// Mitsubishi GX Works2 project: Group13 - Copy   PLC: FX3G

// global labels: Global1
VAR_GLOBAL
  Start_of_Day AT X007 : BOOL;
  Y_0 AT Y000 : BOOL;
  Out_Of_Stock AT M1 : BOOL;
  Emergency_Button AT X005 : BOOL;
  Out_Of_Stock_Hold AT M2 : BOOL;
  Oats_Input AT D1100 : REAL;
  Honey_Input AT D1110 : REAL;
  Protein_Input AT D1120 : REAL;
  Oats_Quantity AT D1130 : REAL;
  Honey_Quantity AT D1140 : REAL;
  Protein_Quanity AT D1150 : REAL;
END_VAR
VAR_GLOBAL CONSTANT
  Oat_Min : REAL := 400;
  Honey_Min : REAL := 160;
  Protein_Min : REAL := 320;
END_VAR
VAR_GLOBAL
  Mixing AT X003 : BOOL;
  Analog_Input_1 AT D8280 : INT;
END_VAR
VAR_GLOBAL CONSTANT
  Normalization : REAL := 400;
END_VAR
VAR_GLOBAL
  Input_1 AT D1200 : REAL;
END_VAR
VAR_GLOBAL CONSTANT
  Regular_Group : REAL := 5.1;
END_VAR
VAR_GLOBAL
  IC_Regular AT M4 : BOOL;
END_VAR
VAR_GLOBAL CONSTANT
  Proteinl_Group : REAL := 5;
END_VAR
VAR_GLOBAL
  IC_Protein AT M5 : BOOL;
  Y_4 AT Y004 : BOOL;
  Y_5 AT Y005 : BOOL;
  TC_0 AT TC0 : BOOL;
END_VAR
VAR_GLOBAL CONSTANT
  Timer_5_Sec : INT := 50;
END_VAR
VAR_GLOBAL
  TS_0 AT TS0 : BOOL;
  Y_3 AT Y003 : BOOL;
END_VAR
VAR_GLOBAL CONSTANT
  Cons_400 : REAL := 400;
  Cons_160 : REAL := 160;
  Cons_120 : REAL := 120;
  Cons_240 : REAL := 240;
  Cons_320 : REAL := 320;
END_VAR
VAR_GLOBAL
  End_Perp AT M7 : BOOL;
  Baking AT X002 : BOOL;
END_VAR
VAR_GLOBAL CONSTANT
  Timer_4_Sec : INT := 40;
END_VAR
VAR_GLOBAL
  TC_2 AT TC2 : BOOL;
  TC_1 AT TC1 : BOOL;
  Y_1 AT Y001 : BOOL;
  Y_2 AT Y002 : BOOL;
  TS_1 AT TS1 : BOOL;
  TS_2 AT TS2 : BOOL;
  Stop_Blinker_Regular AT M8 : BOOL;
  Stop_Blinker_Protein AT M9 : BOOL;
  Blinking AT M10 : BOOL;
  Blinking_1_Timer AT TC3 : BOOL;
END_VAR
VAR_GLOBAL CONSTANT
  Blinking_Timer : INT := 2;
END_VAR
VAR_GLOBAL
  TS_3 AT TS3 : BOOL;
  Blinking_2_Timer AT TC4 : BOOL;
  TS_4 AT TS4 : BOOL;
  Baked AT M11 : BOOL;
  Packing AT X006 : BOOL;
  Start_Packing AT M12 : BOOL;
  Packege_Counter AT CC1 : BOOL;
  Pack_One AT X000 : BOOL;
END_VAR
VAR_GLOBAL CONSTANT
  Pack_8 : WORD := 8;
END_VAR
VAR_GLOBAL
  Package_Container AT D1300 : REAL;
END_VAR
VAR_GLOBAL CONSTANT
  Cons_1 : REAL := 1;
  Normalization_2 : REAL := 40;
END_VAR
VAR_GLOBAL
  Output AT D1400 : REAL;
  Analog_Output AT D8282 : INT;
  Stop_Y4 AT M13 : BOOL;
  Stop_M4 AT M3 : BOOL;
  End_Of_Day AT M6 : BOOL;
END_VAR

// task Task_01 (event TRUE, interval 0, priority 31): POU_01

PROGRAM POU_01
(* structured ladder/FBD written out as ST: instructions are called as NAME(EN, inputs, outputs); _pN, _eN, _tN stand for wires *)
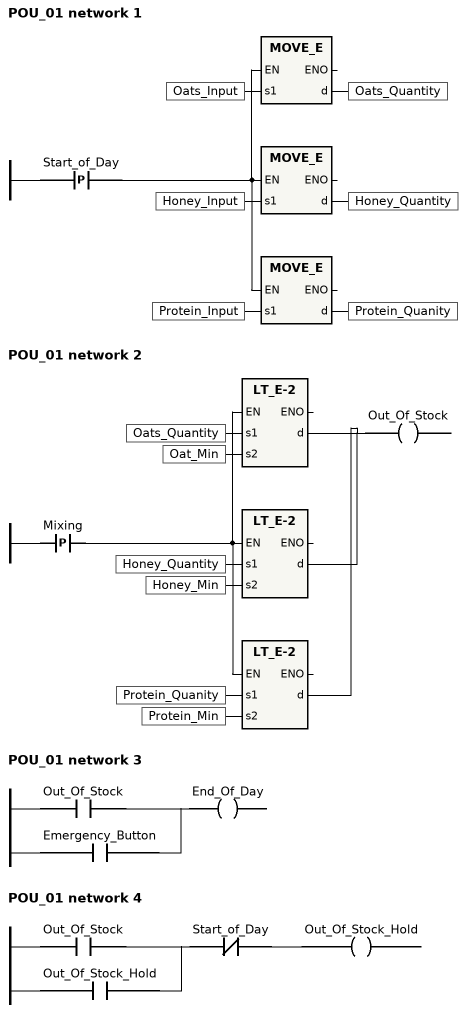
(* network 1 *)
_p1 := LDP(TRUE, Start_of_Day);
MOVE_E(_p1, Oats_Input, Oats_Quantity);
MOVE_E(_p1, Honey_Input, Honey_Quantity);
MOVE_E(_p1, Protein_Input, Protein_Quanity);
(* network 2 *)
_p1 := LDP(TRUE, Mixing);
LT_E(_p1, Oats_Quantity, Oat_Min, _t2);
LT_E(_p1, Honey_Quantity, Honey_Min, _t3);
LT_E(_p1, Protein_Quanity, Protein_Min, _t4);
Out_Of_Stock := _t2 OR _t3 OR _t4;
(* network 3 *)
End_Of_Day := Out_Of_Stock OR Emergency_Button;
(* network 4 *)
Out_Of_Stock_Hold := (Out_Of_Stock OR Out_Of_Stock_Hold) AND NOT Start_of_Day;
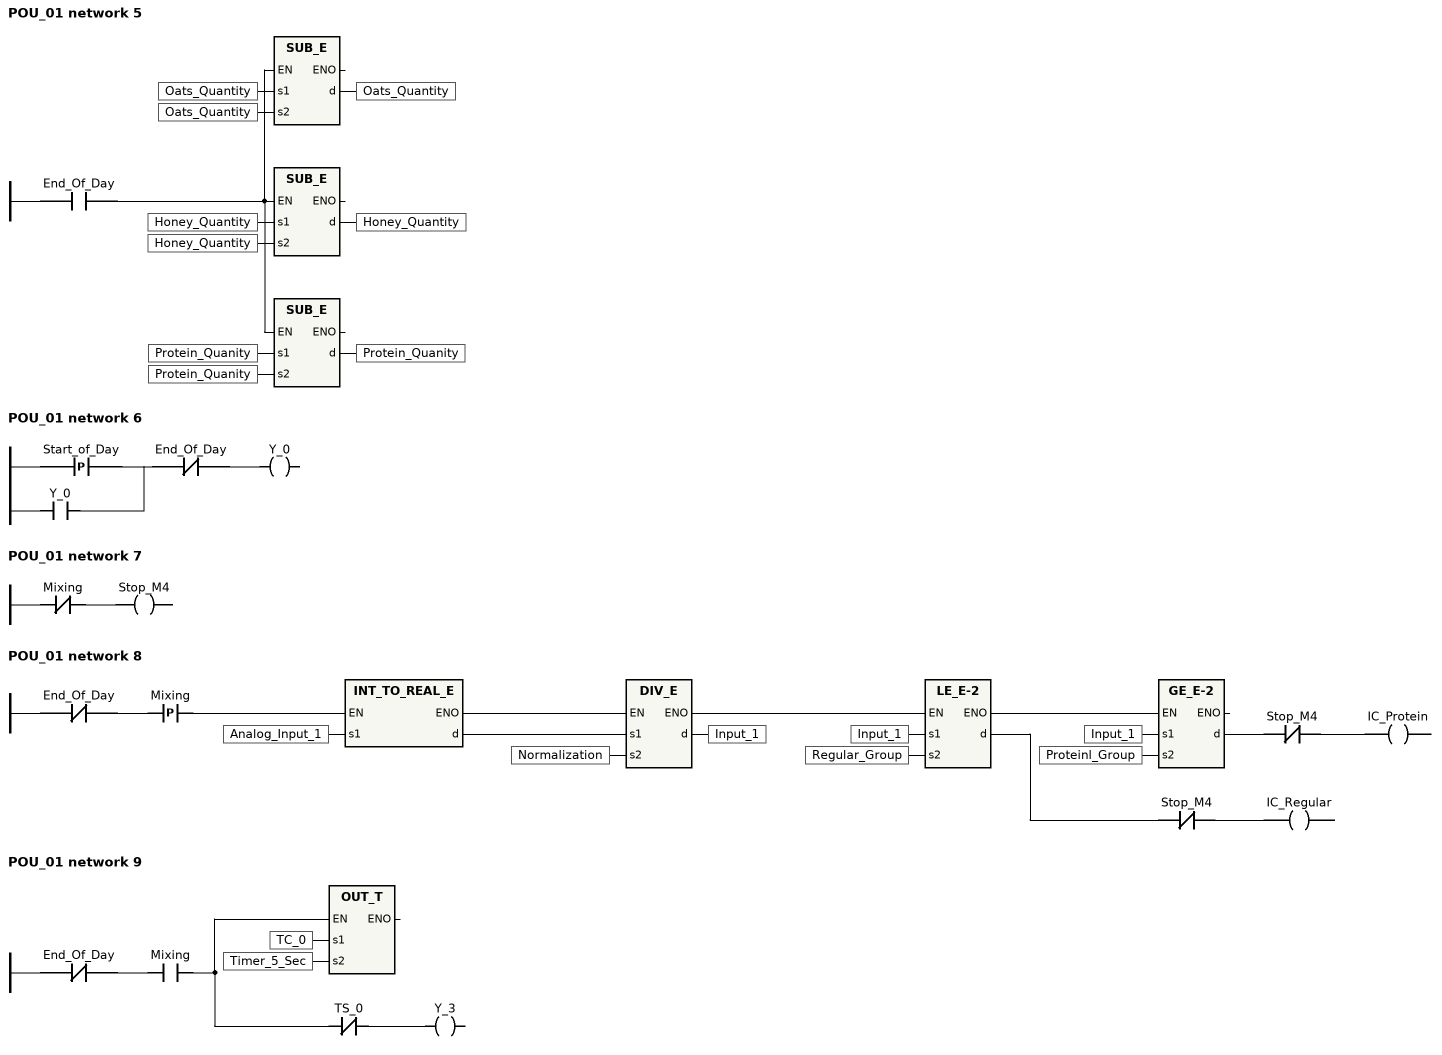
(* network 5 *)
SUB_E(End_Of_Day, Oats_Quantity, Oats_Quantity, Oats_Quantity);
SUB_E(End_Of_Day, Honey_Quantity, Honey_Quantity, Honey_Quantity);
SUB_E(End_Of_Day, Protein_Quanity, Protein_Quanity, Protein_Quanity);
(* network 6 *)
Y_0 := (LDP(TRUE, Start_of_Day) OR Y_0) AND NOT End_Of_Day;
(* network 7 *)
Stop_M4 := NOT Mixing;
(* network 8 *)
_e2 := INT_TO_REAL_E(NOT End_Of_Day AND LDP(TRUE, Mixing), Analog_Input_1, _t1);
_e3 := DIV_E(_e2, _t1, Normalization, Input_1);
_e5 := LE_E(_e3, Input_1, Regular_Group, _t4);
GE_E(_e5, Input_1, Proteinl_Group, _t6);
IC_Protein := _t6 AND NOT Stop_M4;
IC_Regular := _t4 AND NOT Stop_M4;
(* network 9 *)
_p1 := NOT End_Of_Day AND Mixing;
OUT_T(_p1, TC_0, Timer_5_Sec);
Y_3 := _p1 AND NOT TS_0;
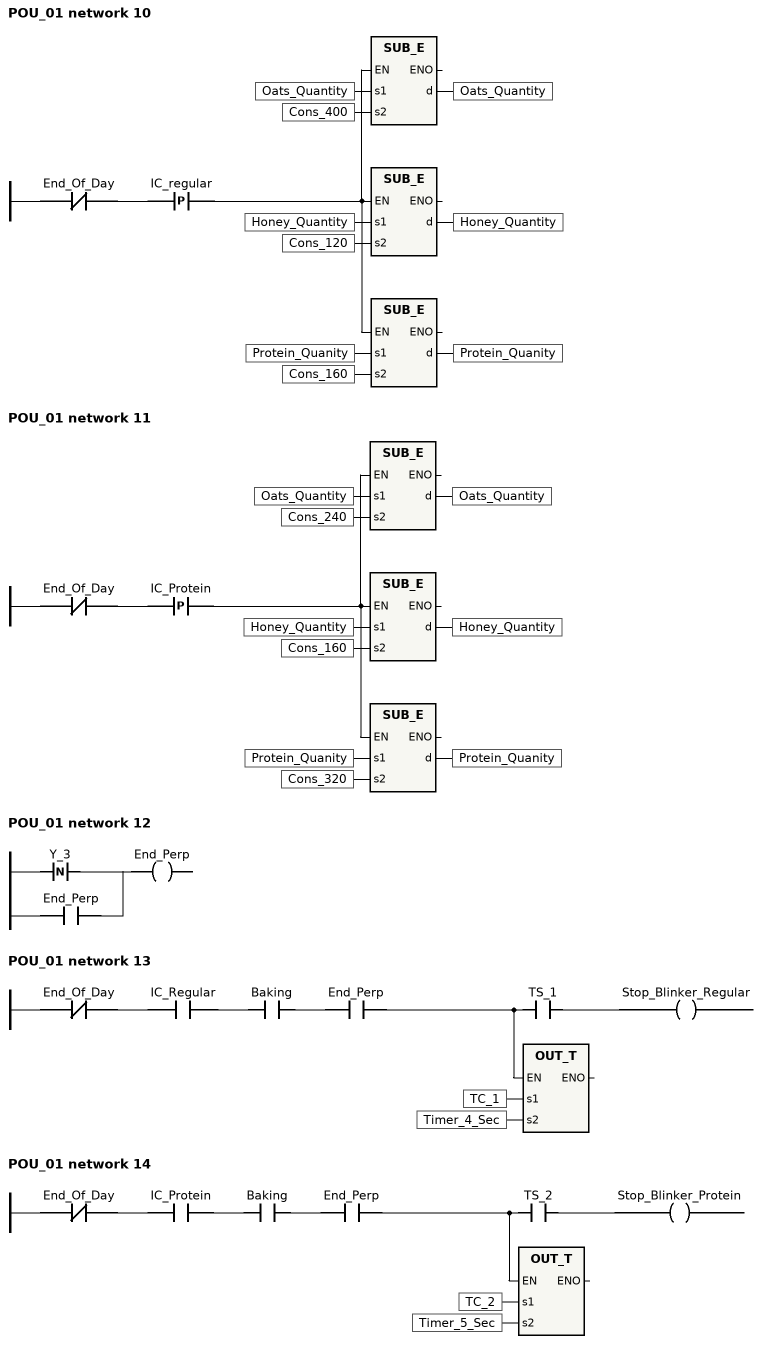
(* network 10 *)
_p1 := NOT End_Of_Day AND LDP(TRUE, IC_regular);
SUB_E(_p1, Oats_Quantity, Cons_400, Oats_Quantity);
SUB_E(_p1, Honey_Quantity, Cons_120, Honey_Quantity);
SUB_E(_p1, Protein_Quanity, Cons_160, Protein_Quanity);
(* network 11 *)
_p1 := NOT End_Of_Day AND LDP(TRUE, IC_Protein);
SUB_E(_p1, Oats_Quantity, Cons_240, Oats_Quantity);
SUB_E(_p1, Honey_Quantity, Cons_160, Honey_Quantity);
SUB_E(_p1, Protein_Quanity, Cons_320, Protein_Quanity);
(* network 12 *)
End_Perp := LDF(TRUE, Y_3) OR End_Perp;
(* network 13 *)
_p1 := NOT End_Of_Day AND IC_Regular AND Baking AND End_Perp;
Stop_Blinker_Regular := _p1 AND TS_1;
OUT_T(_p1, TC_1, Timer_4_Sec);
(* network 14 *)
_p1 := NOT End_Of_Day AND IC_Protein AND Baking AND End_Perp;
Stop_Blinker_Protein := _p1 AND TS_2;
OUT_T(_p1, TC_2, Timer_5_Sec);
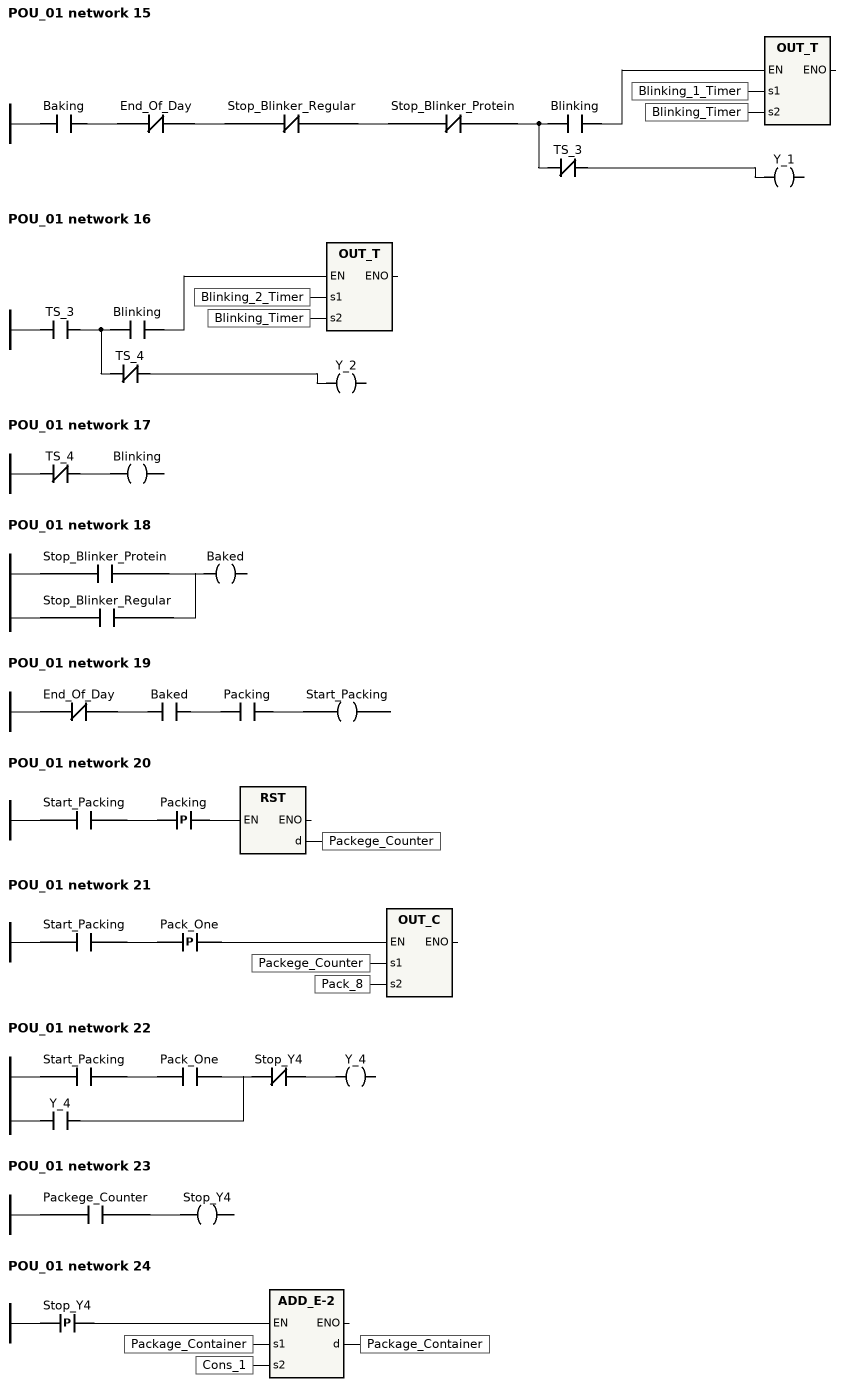
(* network 15 *)
_p1 := Baking AND NOT End_Of_Day AND NOT Stop_Blinker_Regular AND NOT Stop_Blinker_Protein;
OUT_T(_p1 AND Blinking, Blinking_1_Timer, Blinking_Timer);
Y_1 := _p1 AND NOT TS_3;
(* network 16 *)
OUT_T(TS_3 AND Blinking, Blinking_2_Timer, Blinking_Timer);
Y_2 := TS_3 AND NOT TS_4;
(* network 17 *)
Blinking := NOT TS_4;
(* network 18 *)
Baked := Stop_Blinker_Protein OR Stop_Blinker_Regular;
(* network 19 *)
Start_Packing := NOT End_Of_Day AND Baked AND Packing;
(* network 20 *)
RST(Start_Packing AND LDP(TRUE, Packing), Packege_Counter);
(* network 21 *)
OUT_C(Start_Packing AND LDP(TRUE, Pack_One), Packege_Counter, Pack_8);
(* network 22 *)
Y_4 := ((Start_Packing AND Pack_One) OR Y_4) AND NOT Stop_Y4;
(* network 23 *)
Stop_Y4 := Packege_Counter;
(* network 24 *)
ADD_E(LDP(TRUE, Stop_Y4), Package_Container, Cons_1, Package_Container);
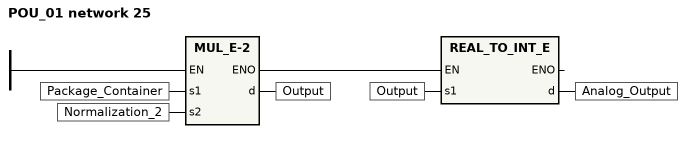
(* network 25 *)
_e1 := MUL_E(TRUE, Package_Container, Normalization_2, Output);
REAL_TO_INT_E(_e1, Output, Analog_Output);
END_PROGRAM
